PROGRAM MAIN
VAR
END_VAR

POU();

END_PROGRAM

(* stored: Version 1.1.0.1, ProductVersion 3.1.4024.3
   POU MAIN: Id {923d4540-8f6f-4f6a-a2d5-ab7087ea5dd7}, SpecialFunc None *)
